FUNCTION CompareReal : BOOL
VAR_INPUT
  value_1: REAL;
  value_2: REAL;
  tolerance: REAL;
END_VAR
VAR
END_VAR

CompareReal := ABS(value_1 - value_2) <= tolerance;

END_FUNCTION

(* stored: Version 1.1.0.1, ProductVersion 3.1.4022.18
   POU CompareReal: Id {d19f00bb-07b3-4d7e-81cd-08b61d36e89f}, SpecialFunc None *)
